{attribute 'qualified_only'}
VAR_GLOBAL
	fSimulationTime : LREAL; 
	bSimulationRunning : BOOL;
	fCylinderVelocity : LREAL;
	fCylinderPosition : LREAL;
	pt0_x : INT := 0;
	pt0_y : INT := 0;
	pt1_x : INT := 0;
	pt1_y : INT; 
	bPistonUpperEndStop : BOOL;
	bPistonLowerEndStop : BOOL;
END_VAR

(* stored: Version 1.1.0.1, ProductVersion 3.1.4024.10
   GVL Outputs: Id {6100726c-2a37-4206-8249-64f2ca6ce4cf} *)
